Staubli VAL3: _writeTxtBoxVal.pgx

program _writeTxtBoxVal(num x_nIndex, num x_nDisplay, string x_sAlign)
  local bool l_bOk
  local num l_nTxtBoxLen
  local string l_sValToDisplay
begin
  // This program displays the content of the selected textbox item
  //
  // Input Param
  //  x_nIndex    : Number of the textbox to display
  //  x_nDisplay : property of the display
  //       =0   : Normal video
  //       =1   : Inverse video
  //       =2   : written in normal video with one selected char inverted
  //  x_sAlign    : text alignment (R=right,L=Left,C=Centered)
  //
  // Output Param
  //  x_Error : Error code
  //
  //Created 21/12/05                              CCUR
  //--------------------------------------------------------------
  // Get length of the string to display
  toNum(pw:sTxtBoxLen[x_nIndex],l_nTxtBoxLen,l_bOk)
  l_sValToDisplay=pw:sTxtBoxVal[x_nIndex]
  call ut:strAlign(l_sValToDisplay,l_nTxtBoxLen,x_sAlign," ")
  gotoxy(nTxtPosX[x_nIndex]+len(pw:sTxtBoxCaption[x_nIndex]),nTxtPosY[x_nIndex])
  switch x_nDisplay
    // Normal video
    case 0
      setTextMode(0)
      //put (pw:sTxtBoxVal[x_nIndex])
      put(l_sValToDisplay)
    break
    // Inverse video
    case 1
      setTextMode(1)
      //put (pw:sTxtBoxVal[x_nIndex])
      put(l_sValToDisplay)
      setTextMode(0)
    break
    // Custom
    case 2
    break
  endSwitch
end
